TYPE ST_ITC_DAR :
(**************************************************************************************
 * 	Application		:	BoxControl Framework
 *	Revision		:	$Revision: 404529 $
 *	Revision date	:	$Date: 2018-04-23 08:21:38 +0200 (Mo., 23 Apr 2018) $
 *	Last changed by	:	$Author: b7bolm $
 *	URL				:	$URL: http://almscdc.swisslog.com/repo/SWPD/Development/BoxControlFramework/20_Release/trunk/01_Software/BCF/BCF/JumpStart/20_Product/10_App/11_Com/10_Lib/10_Conv/11_ITC/01_DUTs/ST_ITC_DAR.TcDUT $
 *
 *	Purpose			:	DAR Structure 					
 *
 *
 * ------------------------------------------------------------------------------------
 *	Copyright Swisslog [IP AG], Switzerland. All rights reserved.
 * 
 * ------------------------------------------------------------------------------------
 *	
 * 	Revision History: 
 *
 * 	VERSION			DATE			INITIALS			DESCRIPTION
 *	0.1				01.01.2001		swl					Example
 *
 **************************************************************************************)	
STRUCT
	Position		: STRING(Conveyor.POSITION_STRINGLENGTH);// 12 Digit SIS Location MM-GGG-EEEE-FF-Z
	Code			: INT;	// Request All = 0 Disable all =1 
	NumberOfSets	: INT;	//Number of Sets to Process in Telegram 
	Set				: ARRAY[E_CM_Index.E_BEGIN_VARIABLE+1..E_CM_Index.E_END_VARIABLE-1] OF ST_CM_Settings;
	SetOffset		: E_CM_Index;	// Offset of Set Number to send 
	eErrorCode		: E_ErrorConv;// 4 Digit error code
END_STRUCT
END_TYPE

(* stored: Version 1.1.0.1, ProductVersion 3.1.4022.12
   DUT ST_ITC_DAR: Id {548f507a-e267-4bdf-912d-e32ff620fc9f} *)
